ABB RobotStudio station: Proyecto_20210527-124155.rsstn

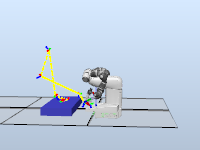
Station Proyecto (saved by RobotStudio 21.1.9443.2)
Controller IRB14000
  mechanical unit ROB_R: IRB14000_0.5_0.5_R, 6 joints, base frame (0, 0, 0) mm
  mechanical unit ROB_R_7: IRB14000_0.5_0.5_R, 1 joints, base frame (0, 0, 0) mm
  mechanical unit ROB_L: IRB14000_0.5_0.5_L, 6 joints, base frame (0, 0, 0) mm
  mechanical unit ROB_L_7: IRB14000_0.5_0.5_L, 1 joints, base frame (0, 0, 0) mm
Layout (positions relative to the parent item):
  - IRB14000_0.5_0.5 [mechanism, from Robots\IRB14000_0.5_0.5__02.rslib] at (0, 0, 0) mm
  - IRB14000_0.5_0.5_R [mechanism, from Robots\IRB14000_0.5_0.5__02.rslib] at (0, 0, 0) mm; joint values [0, -2.2689, -2.3562, 0.5236, 0, 0.6981, -3.1358] (rad or m)
  - IRB14000_0.5_0.5_L [mechanism, from Robots\IRB14000_0.5_0.5__02.rslib] at (0, 0, 0) mm; joint values [0, -2.2689, 2.3562, 0.5236, 0, 0.6981, 0] (rad or m)
  - Part_1 [part] at (462, 0, 0) mm
  - MyTool [mechanism, from Training Objects\myTool.rslib] at (-9.58, -182.61, 198.63) mm, rotated rx 179.99 ry 63.64 rz -165.29 deg
  - Chip [part] at (492.85, 200, 101) mm
  - Drill_holder [mechanism] at (-9.58, 182.61, 198.63) mm, rotated rx -179.34 ry -63.63 rz -15.45 deg; joint values [-0.025, -0.001, -0.0002] (rad or m)
      TCP Tip_holder_mechanism at (-0.08, -53.38, 109.89) mm, rotated rx -73 ry 2 rz -178 deg
      links: L1, L2, L3, L4
  - Part_33 [part] at (486.93, 0, 101) mm, rotated rx 0 ry 0 rz 90 deg
Attachment: MyTool is attached to IRB14000_0.5_0.5_R / Link7
Attachment: Drill_holder is attached to IRB14000_0.5_0.5_L / Link7
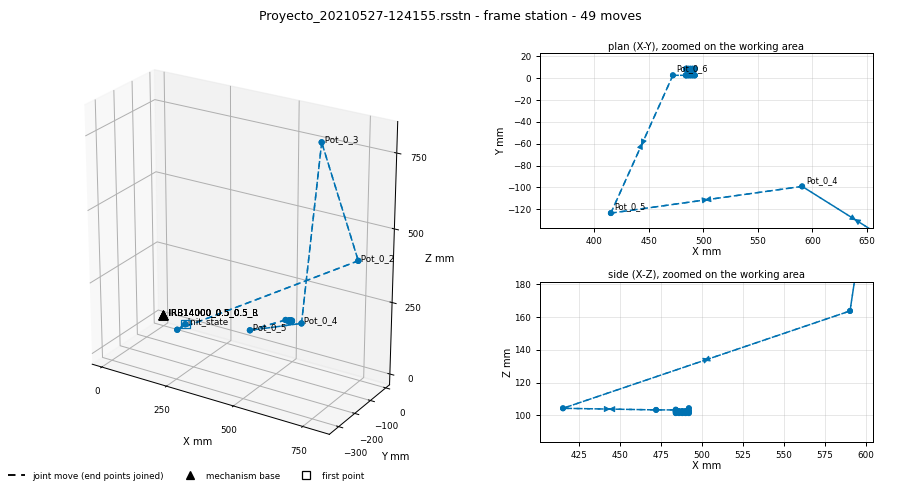
[picture p0: tool path of Proyecto_20210527-124155.rsstn in frame station, 49 of 49 moves have a stored position in this frame; points joined in program order, loops and branches not executed]
Targets, tools, work objects and paths stored in the station, written as RAPID:
! task T_ROB_R
MODULE CalibData
  PERS tooldata MyTool:=[TRUE,[[31.792631019,0,229.638935148],[0.945518576,0,0.325568154,0]],[1,[0,0,1],[1,0,0,0],0,0,0]];
ENDMODULE

! task T_ROB_R
MODULE Module1
  CONST robtarget Init_state:=[[175.771799788,-133.936334157,68.163208612],[0.220019445,-0.124834347,0.967057146,0.028430707],[0,0,-2,4],[-101.964427132,9E+09,9E+09,9E+09,9E+09,9E+09]];
  CONST robtarget Pot_0_1:=[[282.63851741,-340.819698768,162.147776362],[0.105568742,0.881349299,-0.428938056,0.167603097],[0,1,-3,0],[36.752032663,9E+09,9E+09,9E+09,9E+09,9E+09]];
  CONST robtarget Pot_0_2:=[[805.746481197,-131.478847588,443.611196027],[0.093603339,0.75659935,0.398721413,0.509722545],[0,1,-3,0],[17.294413616,9E+09,9E+09,9E+09,9E+09,9E+09]];
  CONST robtarget Pot_0_3:=[[687.671962467,-159.959654994,813.591448779],[0.828352157,0.209765147,0.322982587,0.406833549],[0,1,0,1],[82.238072921,9E+09,9E+09,9E+09,9E+09,9E+09]];
  CONST robtarget Pot_0_4:=[[590.547168499,-98.993259069,163.691697817],[0.335236004,-0.168177429,-0.926608093,0.027029893],[0,0,0,0],[80.11805131,9E+09,9E+09,9E+09,9E+09,9E+09]];
  CONST robtarget Pot_0_5:=[[415.342725267,-123.46779756,104.28687841],[0.522487933,-0.19765224,-0.826763059,0.066353573],[0,0,0,0],[79.453614888,9E+09,9E+09,9E+09,9E+09,9E+09]];
  CONST robtarget Pot_0_6:=[[472.176536102,2.75169226,103.312635348],[0.418722396,-0.063346331,-0.905892526,0.00418673],[1,0,0,0],[86.440027328,9E+09,9E+09,9E+09,9E+09,9E+09]];
  CONST robtarget legr_enter:=[[484.177640449,2.748235942,103.308836916],[0.418725834,-0.063345983,-0.90589095,0.004189096],[1,0,0,0],[86.440027075,9E+09,9E+09,9E+09,9E+09,9E+09]];
  CONST robtarget legr_1_w:=[[484.177845913,2.747723006,101.308341761],[0.418726268,-0.063345905,-0.905890754,0.004189445],[1,0,0,0],[86.440026017,9E+09,9E+09,9E+09,9E+09,9E+09]];
  CONST robtarget legr_1_e:=[[484.177924897,2.747204171,102.307741695],[0.418726788,-0.063345822,-0.905890517,0.004189793],[1,0,0,0],[86.440028939,9E+09,9E+09,9E+09,9E+09,9E+09]];
  CONST robtarget legr_2_e:=[[486.178059863,2.746844936,102.307333468],[0.418727202,-0.063345786,-0.905890328,0.004190036],[1,0,0,0],[86.440024564,9E+09,9E+09,9E+09,9E+09,9E+09]];
  CONST robtarget legr_2_w:=[[486.178145818,2.74666294,101.307134051],[0.418727386,-0.063345778,-0.905890242,0.004190163],[1,0,0,0],[86.440025637,9E+09,9E+09,9E+09,9E+09,9E+09]];
  CONST robtarget legr_3_e:=[[488.178366821,2.746111375,102.306544048],[0.41872787,-0.063345748,-0.905890019,0.004190529],[1,0,0,0],[86.440026029,9E+09,9E+09,9E+09,9E+09,9E+09]];
  CONST robtarget legr_3_w:=[[488.178478351,2.745928708,101.306336227],[0.418728047,-0.063345729,-0.905889938,0.00419065],[1,0,0,0],[86.440025513,9E+09,9E+09,9E+09,9E+09,9E+09]];
  CONST robtarget legr_4_e:=[[490.178651185,2.745459557,102.305739299],[0.418728593,-0.06334561,-0.905889693,0.004190968],[1,0,0,0],[86.440029087,9E+09,9E+09,9E+09,9E+09,9E+09]];
  CONST robtarget legr_4_w:=[[490.178670044,2.745273907,101.305537862],[0.418728757,-0.063345598,-0.905889617,0.004191097],[1,0,0,0],[86.440025193,9E+09,9E+09,9E+09,9E+09,9E+09]];
  CONST robtarget legr_5_e:=[[492.178953648,2.744703279,102.304931071],[0.418729297,-0.063345583,-0.905889366,0.004191471],[1,0,0,0],[86.440022889,9E+09,9E+09,9E+09,9E+09,9E+09]];
  CONST robtarget legr_5_w:=[[492.178940306,2.744532877,101.304739874],[0.418729463,-0.063345549,-0.905889292,0.004191589],[0,0,0,0],[86.440026814,9E+09,9E+09,9E+09,9E+09,9E+09]];
  CONST robtarget legr_exit:=[[492.179250755,2.744140808,104.304432201],[0.418729758,-0.063345547,-0.905889154,0.004191834],[1,0,0,0],[86.440024676,9E+09,9E+09,9E+09,9E+09,9E+09]];
  CONST robtarget legl_enter:=[[492.1792375,8.742008189,104.302027287],[0.418731765,-0.063345285,-0.905888238,0.004193328],[1,0,0,0],[86.440025855,9E+09,9E+09,9E+09,9E+09,9E+09]];
  CONST robtarget legl_1_w:=[[492.180054048,8.739806387,101.499825429],[0.418745915,-0.063330509,-0.905882597,0.00422209],[0,0,0,0],[86.440025476,9E+09,9E+09,9E+09,9E+09,9E+09]];
  CONST robtarget legl_1_e:=[[492.18004979,8.739232692,102.499240164],[0.418746458,-0.063330471,-0.905882347,0.004222475],[0,0,0,0],[86.44002627,9E+09,9E+09,9E+09,9E+09,9E+09]];
  CONST robtarget legl_2_e:=[[490.180259671,8.738864462,102.498840871],[0.418746745,-0.063330421,-0.905882216,0.00422272],[1,0,0,0],[86.440025812,9E+09,9E+09,9E+09,9E+09,9E+09]];
  CONST robtarget legl_2_w:=[[490.180357199,8.738669503,101.498639938],[0.418746921,-0.063330419,-0.905882135,0.00422285],[1,0,0,0],[86.440025935,9E+09,9E+09,9E+09,9E+09,9E+09]];
  CONST robtarget legl_3_e:=[[488.180527467,8.737777912,102.497632429],[0.418747795,-0.063330318,-0.905881735,0.004223488],[1,0,0,0],[86.440028253,9E+09,9E+09,9E+09,9E+09,9E+09]];
  CONST robtarget legl_3_w:=[[488.180525158,8.737612648,101.497439871],[0.418747971,-0.063330287,-0.905881655,0.004223609],[1,0,0,0],[86.440027412,9E+09,9E+09,9E+09,9E+09,9E+09]];
  CONST robtarget legl_4_e:=[[486.180671968,8.737053657,102.496821411],[0.418748431,-0.06333027,-0.905881442,0.004223964],[1,0,0,0],[86.440023469,9E+09,9E+09,9E+09,9E+09,9E+09]];
  CONST robtarget legl_4_w:=[[486.18074824,8.736882674,101.49663065],[0.418748544,-0.063330238,-0.905881391,0.004224077],[1,0,0,0],[86.44002696,9E+09,9E+09,9E+09,9E+09,9E+09]];
  CONST robtarget legl_5_e:=[[484.181019884,8.736350804,102.496027749],[0.41874908,-0.063330147,-0.905881148,0.004224465],[1,0,0,0],[86.440024978,9E+09,9E+09,9E+09,9E+09,9E+09]];
  CONST robtarget legl_5_w:=[[484.181036911,8.736183038,101.495841142],[0.418749233,-0.063330105,-0.90588108,0.004224586],[1,0,0,0],[86.440026654,9E+09,9E+09,9E+09,9E+09,9E+09]];
  CONST robtarget legl_exit:=[[484.181022627,8.735810695,103.495432719],[0.418749593,-0.063330073,-0.905880914,0.00422487],[1,0,0,0],[86.440024977,9E+09,9E+09,9E+09,9E+09,9E+09]];
  PROC main()
    MoveL Init_state,v200,fine,MyTool\WObj:=wobj0;
    MoveJ Pot_0_1,v200,fine,MyTool\WObj:=wobj0;
    MoveJ Pot_0_2,v200,fine,MyTool\WObj:=wobj0;
    MoveJ Pot_0_3,v200,fine,MyTool\WObj:=wobj0;
    MoveJ Pot_0_4,v200,fine,MyTool\WObj:=wobj0;
    MoveJ Pot_0_5,v200,fine,MyTool\WObj:=wobj0;
    MoveJ Pot_0_6,v200,fine,MyTool\WObj:=wobj0;
    MoveJ legr_enter,v200,fine,MyTool\WObj:=wobj0;
    MoveJ legr_1_e,v200,fine,MyTool\WObj:=wobj0;
    MoveJ legr_1_w,v200,fine,MyTool\WObj:=wobj0;
    MoveJ legr_1_e,v200,fine,MyTool\WObj:=wobj0;
    MoveJ legr_2_e,v200,fine,MyTool\WObj:=wobj0;
    MoveJ legr_2_w,v200,fine,MyTool\WObj:=wobj0;
    MoveJ legr_2_e,v200,fine,MyTool\WObj:=wobj0;
    MoveJ legr_3_e,v200,fine,MyTool\WObj:=wobj0;
    MoveJ legr_3_w,v200,fine,MyTool\WObj:=wobj0;
    MoveJ legr_3_e,v200,fine,MyTool\WObj:=wobj0;
    MoveJ legr_4_e,v200,fine,MyTool\WObj:=wobj0;
    MoveJ legr_4_w,v200,fine,MyTool\WObj:=wobj0;
    MoveJ legr_4_e,v200,fine,MyTool\WObj:=wobj0;
    MoveJ legr_5_e,v200,fine,MyTool\WObj:=wobj0;
    MoveJ legr_5_w,v200,fine,MyTool\WObj:=wobj0;
    MoveJ legr_5_e,v200,fine,MyTool\WObj:=wobj0;
    MoveJ legr_exit,v200,fine,MyTool\WObj:=wobj0;
    MoveJ legl_enter,v200,fine,MyTool\WObj:=wobj0;
    MoveJ legl_1_e,v200,fine,MyTool\WObj:=wobj0;
    MoveJ legl_1_w,v200,fine,MyTool\WObj:=wobj0;
    MoveJ legl_1_e,v200,fine,MyTool\WObj:=wobj0;
    MoveJ legl_2_e,v200,fine,MyTool\WObj:=wobj0;
    MoveJ legl_2_w,v200,fine,MyTool\WObj:=wobj0;
    MoveJ legl_2_e,v200,fine,MyTool\WObj:=wobj0;
    MoveJ legl_3_e,v200,fine,MyTool\WObj:=wobj0;
    MoveJ legl_3_w,v200,fine,MyTool\WObj:=wobj0;
    MoveJ legl_3_e,v200,fine,MyTool\WObj:=wobj0;
    MoveJ legl_4_e,v200,fine,MyTool\WObj:=wobj0;
    MoveJ legl_4_w,v200,fine,MyTool\WObj:=wobj0;
    MoveJ legl_4_e,v200,fine,MyTool\WObj:=wobj0;
    MoveJ legl_5_e,v200,fine,MyTool\WObj:=wobj0;
    MoveJ legl_5_w,v200,fine,MyTool\WObj:=wobj0;
    MoveJ legl_5_e,v200,fine,MyTool\WObj:=wobj0;
    MoveJ legl_exit,v200,fine,MyTool\WObj:=wobj0;
    MoveJ legr_enter,v200,fine,MyTool\WObj:=wobj0;
    MoveJ Pot_0_6,v200,fine,MyTool\WObj:=wobj0;
    MoveJ Pot_0_5,v200,fine,MyTool\WObj:=wobj0;
    MoveJ Pot_0_4,v200,fine,MyTool\WObj:=wobj0;
    MoveJ Pot_0_3,v200,fine,MyTool\WObj:=wobj0;
    MoveJ Pot_0_2,v200,fine,MyTool\WObj:=wobj0;
    MoveJ Pot_0_1,v200,fine,MyTool\WObj:=wobj0;
    MoveJ Init_state,v200,fine,MyTool\WObj:=wobj0;
  ENDPROC
ENDMODULE

! task T_ROB_L
MODULE Module1
  CONST robtarget Home:=[[61.480882858,158.400356438,102.243977191],[0.078264412,0.604906798,-0.79132965,-0.041950353],[0,0,-1,4],[101.964427132,9E+09,9E+09,9E+09,9E+09,9E+09]];
ENDMODULE

! task T_ROB_L
MODULE CalibData
  PERS tooldata Tip_holder_mechanism:=[TRUE,[[-0.077,-53.377,109.892],[0.024406608,0.003647592,0.594886456,-0.803430842]],[0.5,[0,1.6,65.9],[1,0,0,0],0,0,0]];
ENDMODULE

